// SIMATIC S7-200 project (STEP 7-Micro/WIN), CPU 221 REL 01.10

SYMBOL_TABLE USER1
sta              I0.0
sto              I0.1
bt_ha            I0.2
ct_duoi          I0.3
ct_tren          I0.4
quay             Q0.0
nang             Q0.1
ha               Q0.2
END_SYMBOL_TABLE

ORGANIZATION_BLOCK MAIN:OB1
TITLE=PROGRAM COMMENTS
BEGIN
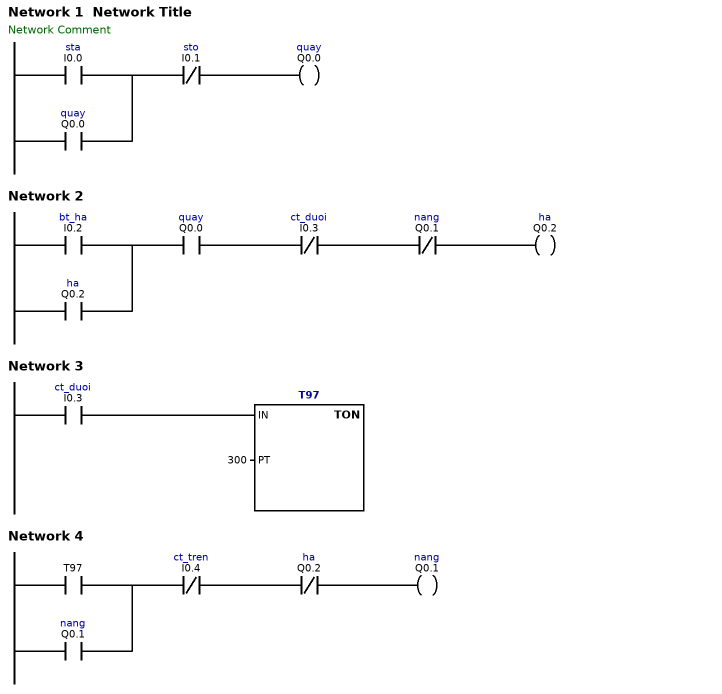
Network 1 // Network Title
// Network Comment
LD     sta:I0.0
O      quay:Q0.0
AN     sto:I0.1
=      quay:Q0.0
Network 2
LD     bt_ha:I0.2
O      ha:Q0.2
A      quay:Q0.0
AN     ct_duoi:I0.3
AN     nang:Q0.1
=      ha:Q0.2
Network 3
LD     ct_duoi:I0.3
TON    T97, 300
Network 4
LD     T97
O      nang:Q0.1
AN     ct_tren:I0.4
AN     ha:Q0.2
=      nang:Q0.1
END_ORGANIZATION_BLOCK
